VISUALIZATION visuSafetyRow  // 600x100
END_VISUALIZATION

(* stored: Version 1.1.0.1, ProductVersion 3.1.4024.12
   Visu visuSafetyRow: Id {3a1b3110-8237-4e7a-b68f-276ccbd63a3e} *)
